FUNCTION_BLOCK FB_PneuCyl_1Pos EXTENDS FB_Base
VAR_INPUT
END_VAR
VAR_OUTPUT
END_VAR
VAR
END_VAR

{error 'Eigenschaftenimplementierung hinzufügen oder Eigenschaft löschen, um die Basisimplementierung zu verwenden'}
PROPERTY Busy : BOOL
GET
END_GET
SET
END_SET
END_PROPERTY

{error 'Eigenschaftenimplementierung hinzufügen oder Eigenschaft löschen, um die Basisimplementierung zu verwenden'}
PROPERTY Done : BOOL
GET
END_GET
SET
END_SET
END_PROPERTY

{error 'Eigenschaftenimplementierung hinzufügen oder Eigenschaft löschen, um die Basisimplementierung zu verwenden'}
PROPERTY Enable : BOOL
GET
END_GET
SET
END_SET
END_PROPERTY

{error 'Eigenschaftenimplementierung hinzufügen oder Eigenschaft löschen, um die Basisimplementierung zu verwenden'}
PROPERTY Error : BOOL
GET
END_GET
SET
END_SET
END_PROPERTY

//FB_Init ist immer implizit verfügbar und wird primär für die Initialisierung verwendet.
//Der Rückgabewert wird nicht ausgewertet. Für gezielte Einflussnahme können Sie
//die Methoden explizit deklarieren und darin mit dem Standard-Initialisierungscode 
//zusätzlichen Code bereitstellen. Sie können den Rückgabewert auswerten.
METHOD FB_Init: BOOL
VAR_INPUT    
	bInitRetains					: BOOL; 					// TRUE: Die Retain-Variablen werden initialisiert (Reset warm / Reset kalt)    
	bInCopyCode						: BOOL;  					// TRUE: Die Instanz wird danach in den Kopiercode kopiert (Online-Change)
	
	I_Name                : STRING;         //  Name
	I_ID                  : UINT;            // ID
END_VAR
END_METHOD

{error 'Eigenschaftenimplementierung hinzufügen oder Eigenschaft löschen, um die Basisimplementierung zu verwenden'}
PROPERTY ID : UINT
GET
END_GET
SET
END_SET
END_PROPERTY

{error 'Methodenimplementierung hinzufügen oder Methode löschen, um die Basisimplementierung zu verwenden'}
METHOD mEnable : BOOL
END_METHOD

{error 'Methodenimplementierung hinzufügen oder Methode löschen, um die Basisimplementierung zu verwenden'}
METHOD mInit : BOOL
END_METHOD

{error 'Eigenschaftenimplementierung hinzufügen oder Eigenschaft löschen, um die Basisimplementierung zu verwenden'}
PROPERTY Mode : E_Mode
GET
END_GET
SET
END_SET
END_PROPERTY

{error 'Methodenimplementierung hinzufügen oder Methode löschen, um die Basisimplementierung zu verwenden'}
METHOD mReset : BOOL
END_METHOD

{error 'Eigenschaftenimplementierung hinzufügen oder Eigenschaft löschen, um die Basisimplementierung zu verwenden'}
PROPERTY Name : STRING
GET
END_GET
SET
END_SET
END_PROPERTY

END_FUNCTION_BLOCK

(* stored: Version 1.1.0.1, ProductVersion 3.1.4026.18
   POU FB_PneuCyl_1Pos: Id {a7b52489-8306-4768-bce5-7bb6030c1e74}, SpecialFunc None
   Folder 01 Properties: Id {c888f04d-257a-4261-96a3-2bc2ced9cf8a}
   Folder 02 Methodes: Id {a74a2467-4e6f-4a46-b8d2-e35efb4de658}
   Property Busy: Id {e580c84e-b274-4f1c-9942-605e02480dcb}
   Get Get: Id {0bdc067b-203b-4007-b07f-9fbbc24101e1}
   Set Set: Id {74170e3a-f218-473d-879b-b312250d3d8d}
   Property Done: Id {843e882c-3ac9-405b-b0b9-910d7a537772}
   Get Get: Id {f87b0759-5c4c-4f3c-bbb8-43573a8ec162}
   Set Set: Id {57f52870-a917-4d54-8f72-4b9f627bcb85}
   Property Enable: Id {050e17ca-282c-4e06-b630-7667ffc73d78}
   Get Get: Id {27d89eaf-1591-41f2-bc3b-6f43f759e320}
   Set Set: Id {77de8c84-c0ab-4551-9c0d-5f01fa0b15c9}
   Property Error: Id {cab2b3b0-4833-4a26-9b3a-875db2d4109d}
   Get Get: Id {2479d3f4-286a-4bbc-b76c-6d181eaa3d75}
   Set Set: Id {37b4aa2a-d320-4c61-b7fd-0e9af1a32822}
   Method FB_Init: Id {34a01689-1654-4ffa-b208-161dc9b86395}
   Property ID: Id {48421c43-54ec-4272-8829-102bb54c8894}
   Get Get: Id {99aef2e9-0e2c-4169-8cac-4c38178b3fbb}
   Set Set: Id {41b850d8-6142-4622-990b-21a4e54bf64b}
   Method mEnable: Id {a837f753-93ae-4f1c-8c43-13d31a0e418c}
   Method mInit: Id {e5d1dcd0-82ba-457b-a512-ca925612ad74}
   Property Mode: Id {967c651f-5ff2-4570-8307-b32955360277}
   Get Get: Id {e33cb558-dced-42b5-83a7-156b180e5cbf}
   Set Set: Id {dabef150-037d-4592-b8f5-4e11fbcefdab}
   Method mReset: Id {bc3e8d40-9767-4b8c-b096-08af42010a51}
   Property Name: Id {73f577ad-4be0-4fe0-9dba-b0591e6ffebc}
   Get Get: Id {3fc94e22-2d91-4b44-b472-95d70d549c73}
   Set Set: Id {c40b8545-966f-429c-92a4-65f9bbd5a20f} *)
